FUNCTION_BLOCK FB_VirtualControlBox IMPLEMENTS I_CraneControlBox
VAR_INPUT
END_VAR
VAR_OUTPUT
END_VAR
VAR
	stCranHMIVaribels		: REFERENCE TO ST_CraneHMIData; // From FB_Init
END_VAR

METHOD FB_init : BOOL
VAR_INPUT
	bInitRetains : BOOL; // if TRUE, the retain variables are initialized (warm start / cold start)
	bInCopyCode : BOOL;  // if TRUE, the instance afterwards gets moved into the copy code (online change)
	stCranHMIVaribelsInit		: REFERENCE TO ST_CraneHMIData;
END_VAR
stCranHMIVaribels := stCranHMIVaribelsInit;
END_METHOD

{warning 'add method implementation '}
METHOD Joystick : REAL
END_METHOD

{warning 'add method implementation '}
METHOD Mode : E_ControlBoxMode
END_METHOD

{warning 'add method implementation '}
METHOD Status : E_RunningStates
END_METHOD

END_FUNCTION_BLOCK

(* stored: Version 1.1.0.1, ProductVersion 3.1.4024.12
   POU FB_VirtualControlBox: Id {622528cd-5650-44d7-9bcf-28eeafb53948}, SpecialFunc None
   Method FB_init: Id {0a9ddb92-dacb-4127-a790-6299cfde9db9}
   Method Joystick: Id {5ea5c0dd-9f95-49a5-908c-6a7dd1b9a81a}
   Method Mode: Id {3b20504c-eddc-4766-aee1-8ca5506d6f63}
   Method Status: Id {3b669f13-e677-405d-846b-051f4ce97bbc} *)
